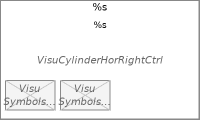
VISUALIZATION VisuCylinderHorRight  // 200x120
VAR_IN_OUT
	fbVisuCylinder: FB_VISU_CYLINDER;
END_VAR
    Textfield (0,15 200x20), "%s", text variable: fbVisuCylinder.strInfo, colour toggle: fbVisuCylinder.stEvent.bEventActive
    Textfield (0,0 200x14), "%s", text variable: fbVisuCylinder.strFullObjName
    Image (60,80 50x30), invisible if: fbVisuCylinder.bWorkArrowInvisible, image: VisuSymbols.Symbols.ArrowBoldRight
        p2175578022: fbVisuCylinder.dwFrameColorWork
    Image (5,80 50x30), invisible if: fbVisuCylinder.bBaseArrowInvisible, image: VisuSymbols.Symbols.ArrowBoldLeft
        p2175578022: fbVisuCylinder.dwFrameColorBase
    Group (5,30 100x40)
        p3560616238: fbVisuCylinder.iNegMove
        RoundedRectangle (0,10 100x20)
        RoundedRectangle (0,0 20x40)
    Rectangle (0,30 100x40)
        OnMouseClick: execute { fbVisuCylinder.bFrameInvisible:=false; }
    Frame (0,0 200x120), invisible if: fbVisuCylinder.bFrameInvisible, frame switch variable: fbVisuCylinder.iFrame
        shows VisuCylinderHorRightCtrl(fbVisuCylinder := fbVisuCylinder)
END_VISUALIZATION

(* stored: Version 1.1.0.1, ProductVersion 3.1.4024.12
   Visu VisuCylinderHorRight: Id {1f762bed-9048-4b02-8a4f-e210c1c900ca} *)
